{attribute addProperty BoxType "EL3773-0000-0017"}
{attribute addProperty Id "Cycle_CountAT %I*UINT162"}
{attribute addProperty CRC "2363401108"}
{attribute addProperty SizeInBites "16"}
{attribute addProperty SizeInBytes "2"}
TYPE AI_Sample_Count_8CDEA394 :
STRUCT
	{attribute addProperty Name "Cycle_Count"}
	Cycle_Count AT %I* : UINT;
END_STRUCT
END_TYPE

(* stored: Version 1.2.0.0, ProductVersion 3.1.4024.9
   DUT AI_Sample_Count_8CDEA394: Id {8a38335e-cd52-4631-ac82-a886abfbe66d} *)
